{attribute 'qualified_only'}
{attribute 'strict'}
TYPE eTcaPushButtonLightState :
(
	none := 0,
	permanent := 1,
	intervall := 2
);
END_TYPE

(* stored: Version 1.1.0.1
   DUT eTcaPushButtonLightState: Id {c274886c-0822-437e-b438-76a1afa23fdf} *)
